{attribute 'GeneratedUsingTerminal: EK1100-0000-0018'}
{attribute addProperty BoxType "EK1100-0000-0018"}
{attribute addProperty Id "Beckhoff_ER5xxxEK1122Beckhoff_ER5xxxEK1122_6E7A8561104"}
{attribute addProperty CRC "3116710967"}
{attribute addProperty Size "104"}
TYPE Beckhoff_ER5xxx_B9C53C37 EXTENDS EK1100_AB5A9467 :
STRUCT
	{attribute addProperty Name "Beckhoff_ER5xxxEK1122"}
	{attribute addProperty PreviousPort "Beckhoff ER5xxx : B"}
	Beckhoff_ER5xxxEK1122 : Beckhoff_ER5xxxEK1122_6E7A8561;
END_STRUCT
END_TYPE

(* stored: Version 1.2.0.0, ProductVersion 3.1.4024.9
   DUT Beckhoff_ER5xxx_B9C53C37: Id {0a899f19-fb75-4a8b-804d-2a7279ea4e04} *)
